// TIA Portal V15.1 export
// export: Created 2024-06-21T08:41:11.8726423Z, ExportSetting WithDefaults, DisplayName Totally Integrated Automation Portal, DisplayVersion V15.1 Update 5, DisplayName TIA Portal Openness, DisplayVersion V15.1 Update 5, DisplayName SINAMICS Startdrive Advanced, DisplayVersion V15.1, DisplayName G130, G150, S120, S150, SINAMICS MV, S210, DisplayVersion V15.1, DisplayName G110M, G120, G120C, G120D, G120P, DisplayVersion V15.1, DisplayName STEP 7 Professional, DisplayVersion V15.1 Update 5, DisplayName STEP 7 Safety, DisplayVersion V15.1, DisplayName WinCC Professional, DisplayVersion V15.1 Update 5, DisplayName SIMATIC Visualization Architect, DisplayVersion V15.1
FUNCTION_BLOCK "LGBRdWrData"   // FB6668, FBD
TITLE = PTC_RdWrData
{ S7_Optimized_Access := 'TRUE' }
VERSION : 0.1
// This module handles the reading and writing of data with indexing.
// It retrigger the index if communication fault or overtime from the same index 
// is active
// stored: AutoNumber false, IsIECCheckEnabled false, IsRetainMemResEnabled false, MemoryReserve 100, SetENOAutomatically False, UDAEnableTagReadback false
   VAR_INPUT
      I_Index { ExternalAccessible := 'False'; ExternalVisible := 'False'; ExternalWritable := 'False'} : Int;   // Index active
      I_IndexStart { ExternalAccessible := 'False'; ExternalVisible := 'False'; ExternalWritable := 'False'} : Int;   // Index start position
      I_IndexEnd { ExternalAccessible := 'False'; ExternalVisible := 'False'; ExternalWritable := 'False'} : Int;   // Index end position
      C_CheckTime { ExternalAccessible := 'False'; ExternalVisible := 'False'; ExternalWritable := 'False'} : DInt;   // Checktime
      C_EnableWrite { ExternalAccessible := 'False'; ExternalVisible := 'False'; ExternalWritable := 'False'} : Bool;   // Enable writing
      C_EnableRead { ExternalAccessible := 'False'; ExternalVisible := 'False'; ExternalWritable := 'False'} : Bool;   // Enable reading
   END_VAR
   VAR_OUTPUT
      O_Read { ExternalAccessible := 'False'; ExternalVisible := 'False'; ExternalWritable := 'False'} : Bool;   // Read position
      O_Write { ExternalAccessible := 'False'; ExternalVisible := 'False'; ExternalWritable := 'False'} : Bool;   // Write position
      O_Index { ExternalAccessible := 'False'; ExternalVisible := 'False'; ExternalWritable := 'False'} : Int;   // Index write or read
   END_VAR
   VAR_IN_OUT
      IO_Done { ExternalAccessible := 'False'; ExternalVisible := 'False'; ExternalWritable := 'False'} : Bool;   // Reading or Writing done
   END_VAR
   VAR
      TimerResult { ExternalAccessible := 'False'; ExternalVisible := 'False'; ExternalWritable := 'False'} : Bool;   // Timer result active
      Read { ExternalAccessible := 'False'; ExternalVisible := 'False'; ExternalWritable := 'False'} : Bool;
      Write { ExternalAccessible := 'False'; ExternalVisible := 'False'; ExternalWritable := 'False'} : Bool;
      TimerValue { ExternalAccessible := 'False'; ExternalVisible := 'False'; ExternalWritable := 'False'} : DInt;   // Active timer value
      CheckTimer { ExternalAccessible := 'False'; ExternalVisible := 'False'; ExternalWritable := 'False'} : "LTimer";
      IndexOld { ExternalAccessible := 'False'; ExternalVisible := 'False'; ExternalWritable := 'False'} : Int;
      IndexOut { ExternalAccessible := 'False'; ExternalVisible := 'False'; ExternalWritable := 'False'} : Int;
   END_VAR
   VAR_TEMP
      ret : Int;
   END_VAR
   VAR_TEMP   // added for the SCL form of the ladder/FBD networks
      _w1 : Bool;
   END_VAR
BEGIN

REGION Network 1: **** 1 - Inputs ****
   // Check overtime o new index
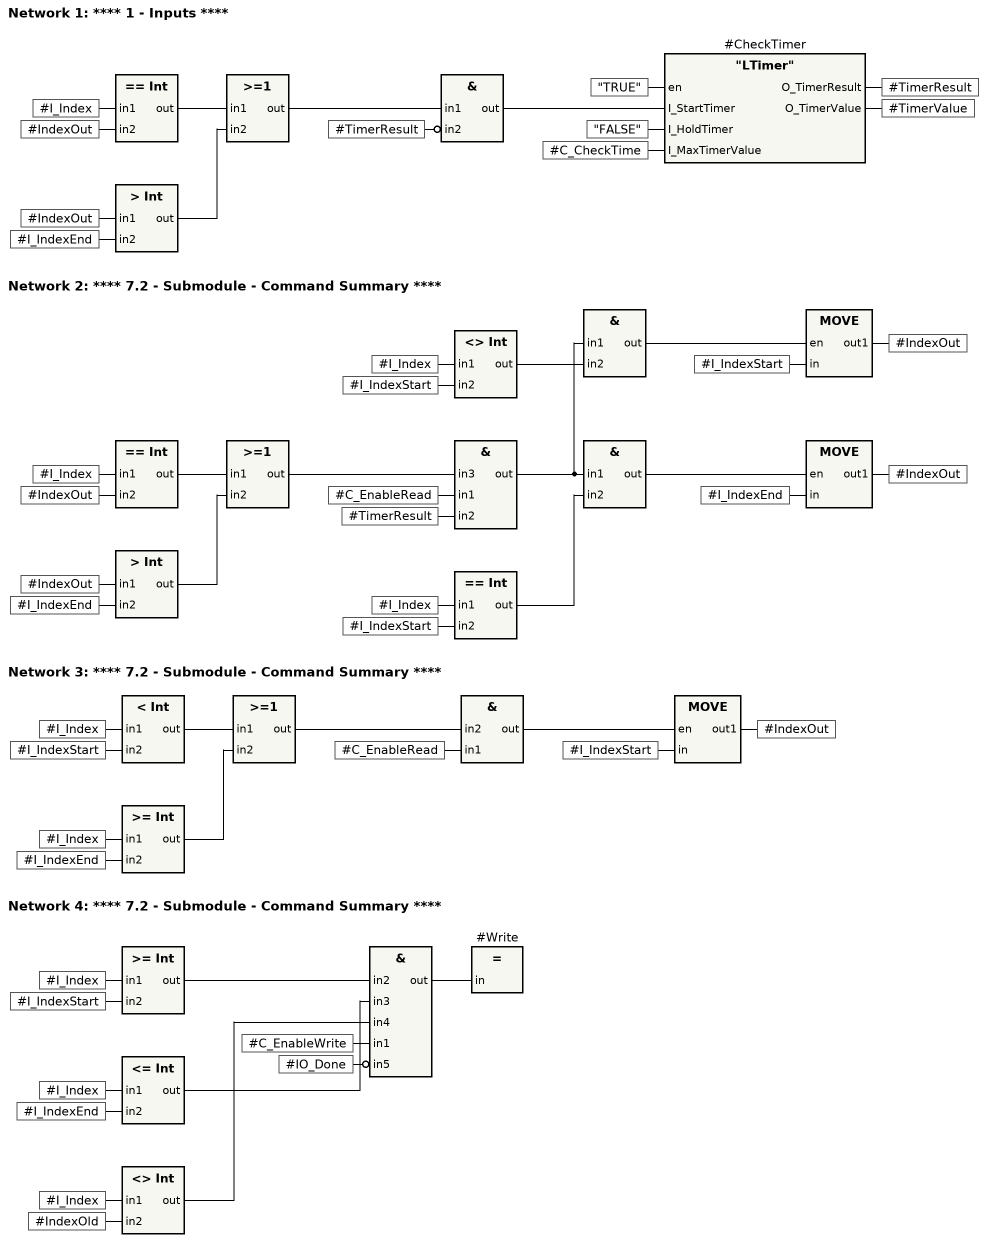
   IF "TRUE" THEN
       #CheckTimer(I_StartTimer := ((#I_Index = #IndexOut) OR (#IndexOut > #I_IndexEnd)) AND NOT #TimerResult,   // "LTimer"
                   I_HoldTimer := "FALSE",
                   I_MaxTimerValue := #C_CheckTime,
                   O_TimerResult => #TimerResult,
                   O_TimerValue => #TimerValue);
   END_IF;
END_REGION

REGION Network 2: **** 7.2 - Submodule - Command Summary ****
   // Retrigger index
   #_w1 := ((#I_Index = #IndexOut) OR (#IndexOut > #I_IndexEnd)) AND #C_EnableRead AND #TimerResult;
   IF #_w1 AND (#I_Index <> #I_IndexStart) THEN #IndexOut := #I_IndexStart; END_IF;
   IF #_w1 AND (#I_Index = #I_IndexStart) THEN #IndexOut := #I_IndexEnd; END_IF;
END_REGION

REGION Network 3: **** 7.2 - Submodule - Command Summary ****
   // Set to startposition
   IF ((#I_Index < #I_IndexStart) OR (#I_Index >= #I_IndexEnd)) AND #C_EnableRead THEN
       #IndexOut := #I_IndexStart;
   END_IF;
END_REGION

REGION Network 4: **** 7.2 - Submodule - Command Summary ****
   // Write position to
   #Write := (#I_Index >= #I_IndexStart) AND (#I_Index <= #I_IndexEnd) AND (#I_Index <> #IndexOld) AND #C_EnableWrite AND NOT #IO_Done;
END_REGION

REGION Network 5: **** 7.2 - Submodule - Command Summary ****
   // Write position to
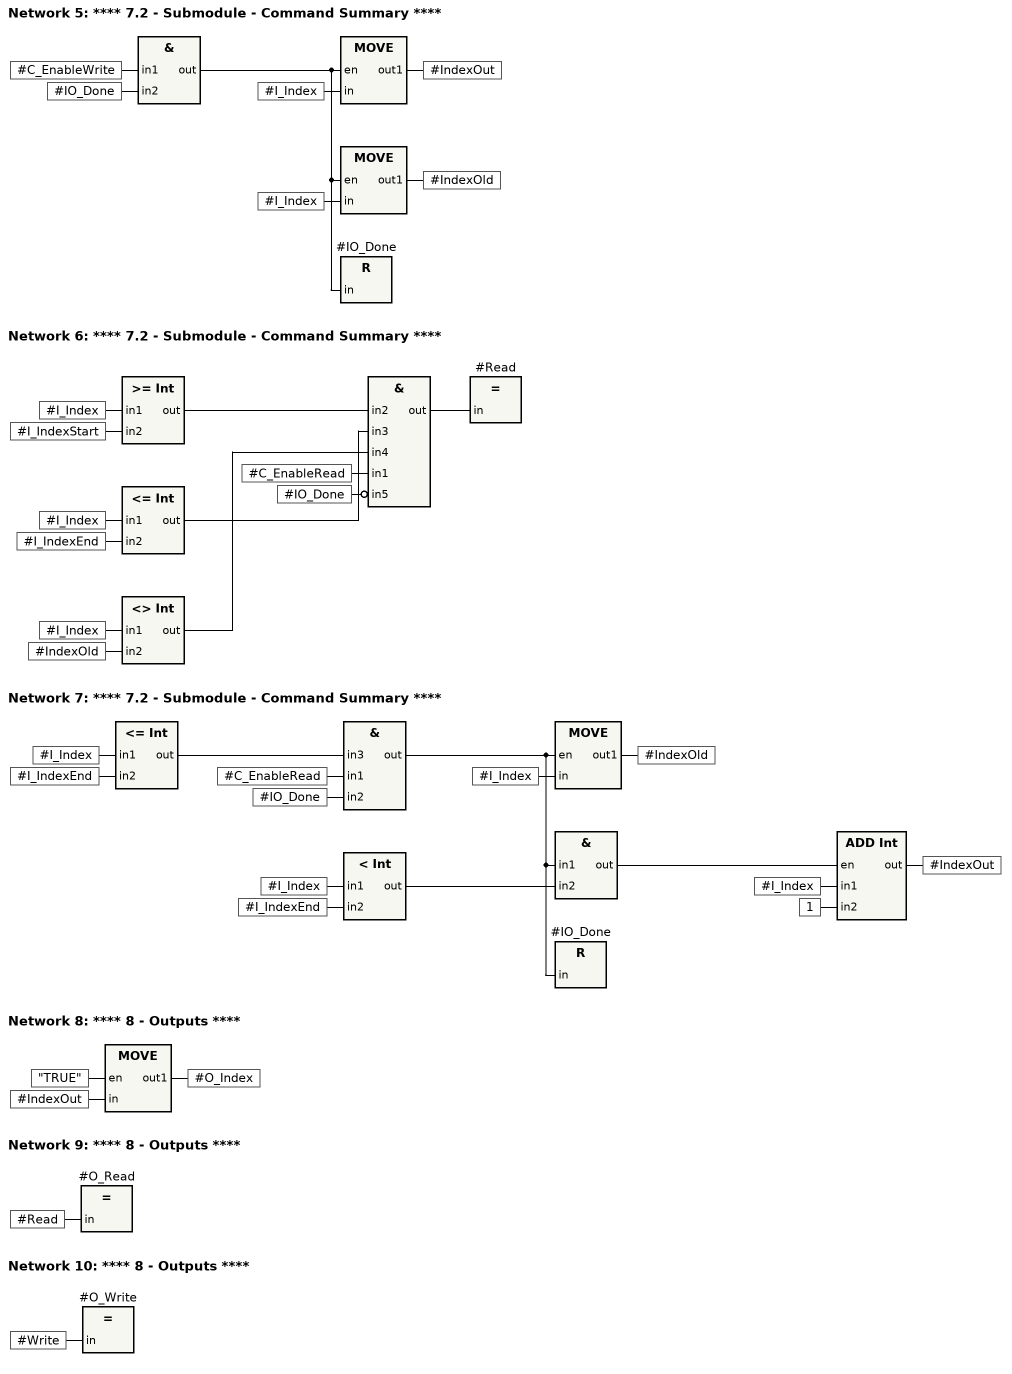
   IF #C_EnableWrite AND #IO_Done THEN
       #IndexOut := #I_Index;
       #IndexOld := #I_Index;
       #IO_Done := FALSE;
   END_IF;
END_REGION

REGION Network 6: **** 7.2 - Submodule - Command Summary ****
   // Read position to
   #Read := (#I_Index >= #I_IndexStart) AND (#I_Index <= #I_IndexEnd) AND (#I_Index <> #IndexOld) AND #C_EnableRead AND NOT #IO_Done;
END_REGION

REGION Network 7: **** 7.2 - Submodule - Command Summary ****
   // Read position to
   #_w1 := (#I_Index <= #I_IndexEnd) AND #C_EnableRead AND #IO_Done;
   IF #_w1 THEN #IndexOld := #I_Index; END_IF;
   IF #_w1 AND (#I_Index < #I_IndexEnd) THEN #IndexOut := #I_Index + 1; END_IF;
   IF #_w1 THEN #IO_Done := FALSE; END_IF;
END_REGION

REGION Network 8: **** 8 - Outputs ****
   // Index Out
   IF "TRUE" THEN #O_Index := #IndexOut; END_IF;
END_REGION

REGION Network 9: **** 8 - Outputs ****
   // Read
   #O_Read := #Read;
END_REGION

REGION Network 10: **** 8 - Outputs ****
   // Write
   #O_Write := #Write;
END_REGION
END_FUNCTION_BLOCK
